(* PLC project Generated.project, CODESYS CODESYS V3.5 SP19 Patch 1 *)
(* stored: creationDateTime 2026-09-20T18:55:02.683253, modificationDateTime 2026-09-20T18:55:02.683253 *)

(* values of E_CycleSampleCountResetMode: NEVER: Defaut : RAZ manuelle IHM uniquement (comportement historique, aucun changement); ON_FIRST_START: RAZ au premier demarrage de cycle apres mise sous tension de l'automate; ON_SAFETY_REARM: RAZ au rearmement de la chaine AU (contacteur puissance reengage) *)

{attribute 'qualified_only'}
{attribute 'strict'}
TYPE E_CycleSampleCountResetMode : (NEVER := 0, ON_FIRST_START := 1, ON_SAFETY_REARM := 2);
END_TYPE
